TYPE ST_GCLiftPinAxisMoveAbsParam :
STRUCT
	Position : LREAL;
	Velocity : LREAL;
	Acceleration : LREAL;
	Deceleration : LREAL;
END_STRUCT
END_TYPE

(* stored: Version 1.1.0.1, ProductVersion 3.1.4026.18
   DUT ST_GCLiftPinAxisMoveAbsParam: Id {4eb5033d-e25a-4e2f-a0c6-a2c41779a1a2} *)
